% RSLogix 500 project LAB05_BAK001.RSS, saved by version 12.00.00.00 %
PROJECT "LAB05"    % processor: MicroLogix 1400 %

PROGRAM FILES
  LAD 2   6 rungs

DATA FILES
  O0 OUTPUT  6 elements
  I1 INPUT  8 elements
  S2 STATUS  66 elements
  B3 BINARY  1 elements
  T4 TIMER  1 elements
  C5 COUNTER  1 elements
  R6 CONTROL  1 elements
  N7 INTEGER  1 elements
  F8 FLOAT  1 elements

LADDER 2
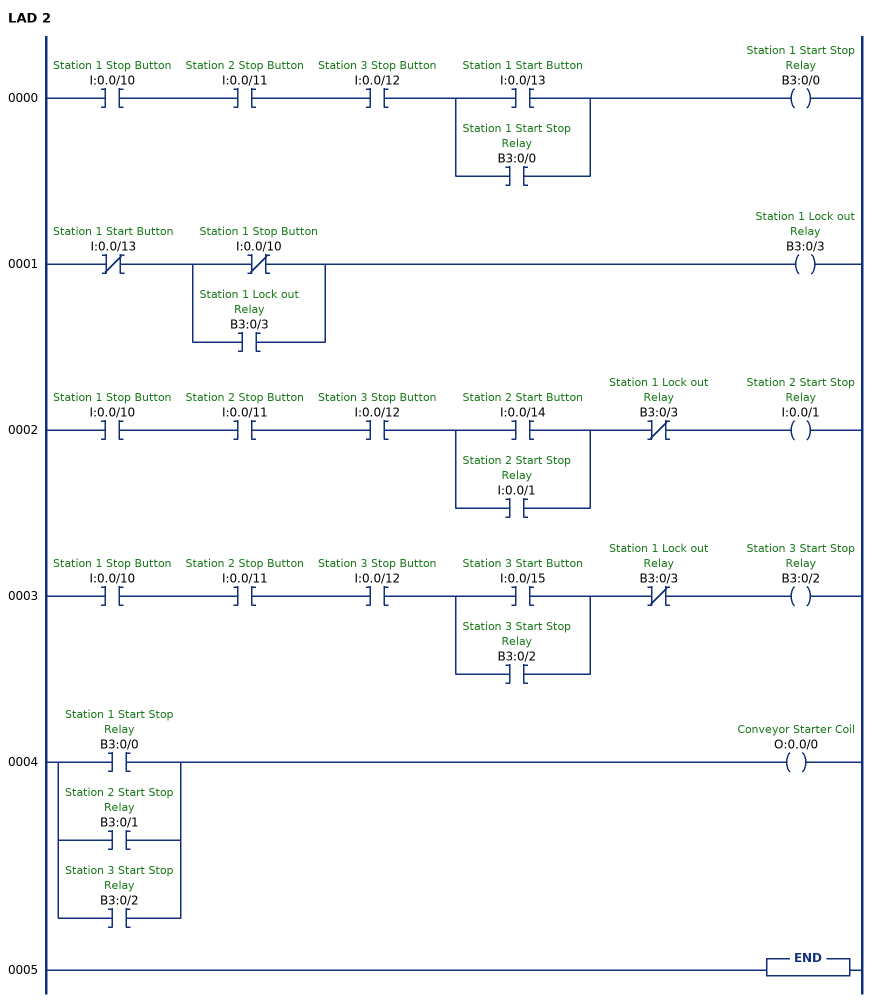
% Rung: 0 %
SOR XIC I:0.0/10 XIC I:0.0/11 XIC I:0.0/12 BST XIC I:0.0/13 NXB XIC B3:0/0 BND OTE B3:0/0 EOR
%   I:0.0/10  "Station 1 Stop Button" %
%   I:0.0/11  "Station 2 Stop Button" %
%   I:0.0/12  "Station 3 Stop Button" %
%   I:0.0/13  "Station 1 Start Button" %
%   B3:0/0  "Station 1 Start Stop Relay" %
% Rung: 1 %
SOR XIO I:0.0/13 BST XIO I:0.0/10 NXB XIC B3:0/3 BND OTE B3:0/3 EOR
%   I:0.0/13  "Station 1 Start Button" %
%   I:0.0/10  "Station 1 Stop Button" %
%   B3:0/3  "Station 1 Lock out Relay" %
% Rung: 2 %
SOR XIC I:0.0/10 XIC I:0.0/11 XIC I:0.0/12 BST XIC I:0.0/14 NXB XIC I:0.0/1 BND XIO B3:0/3 OTE I:0.0/1 EOR
%   I:0.0/10  "Station 1 Stop Button" %
%   I:0.0/11  "Station 2 Stop Button" %
%   I:0.0/12  "Station 3 Stop Button" %
%   I:0.0/14  "Station 2 Start Button" %
%   I:0.0/1  "Station 2 Start Stop Relay" %
%   B3:0/3  "Station 1 Lock out Relay" %
% Rung: 3 %
SOR XIC I:0.0/10 XIC I:0.0/11 XIC I:0.0/12 BST XIC I:0.0/15 NXB XIC B3:0/2 BND XIO B3:0/3 OTE B3:0/2 EOR
%   I:0.0/10  "Station 1 Stop Button" %
%   I:0.0/11  "Station 2 Stop Button" %
%   I:0.0/12  "Station 3 Stop Button" %
%   I:0.0/15  "Station 3 Start Button" %
%   B3:0/2  "Station 3 Start Stop Relay" %
%   B3:0/3  "Station 1 Lock out Relay" %
% Rung: 4 %
SOR BST XIC B3:0/0 NXB BST XIC B3:0/1 NXB XIC B3:0/2 BND BND OTE O:0.0/0 EOR
%   B3:0/0  "Station 1 Start Stop Relay" %
%   B3:0/1  "Station 2 Start Stop Relay" %
%   B3:0/2  "Station 3 Start Stop Relay" %
%   O:0.0/0  "Conveyor Starter Coil" %
% Rung: 5 %
SOR END EOR
